{attribute 'GeneratedUsingTerminal: EP1122-0001-0016'}
{attribute addProperty BoxType "EP1122-0001-0016"}
{attribute addProperty Id "A_0025_EP1122_0001_0017A_0025_EP1122_0001_0017_F097A3BA1330"}
{attribute addProperty CRC "3779772506"}
{attribute addProperty Size "1330"}
TYPE A_0024_EP1122_0001_0016_E14AC05A EXTENDS EP1122_1FC0878B :
STRUCT
	{attribute addProperty Name "A_0025_EP1122_0001_0017"}
	{attribute addProperty PreviousPort "A_0024(EP1122-0001-0016) : D"}
	A_0025_EP1122_0001_0017 : A_0025_EP1122_0001_0017_F097A3BA;
END_STRUCT
END_TYPE

(* stored: Version 1.2.0.0, ProductVersion 3.1.4024.9
   DUT A_0024_EP1122_0001_0016_E14AC05A: Id {32a34a17-506b-464e-9d60-782bedb2f864} *)
